{attribute 'GeneratedUsingTerminal: EK1122-0000-0018'}
{attribute addProperty BoxType "EK1122-0000-0018"}
{attribute addProperty Id "Beckhoff_EP5xxxsub_EK1100EK1100_1FC0878B2A_0001_EP5001_0002_0016EP5001_0B28D08722A_0002_EP5101_0002_0016EP5101_87AC78CF32A_0003_EP5101_0002_0017EP5101_87AC78CF32A_0004_EP5101_0002_0018EP5101_87AC78CF32A_0005_EP5101_0002_0019EP5101_87AC78CF32A_0006_EP5101_0011_0016EP5101_7476E94838A_0007_EP5101_0011_0017EP5101_7476E94838A_0008_EP5101_0011_0018EP5101_7476E94838A_0009_EP5101_0011_0019EP5101_7476E94838A_0010_EP5101_1002_0017EP5101_87AC78CF32A_0011_EP5151_0002_0018EP5151_7476E94838A_0012_EP5101_2011_0016EP5101_382A92AF35"}
{attribute addProperty CRC "1751390652"}
{attribute addProperty Size "409"}
TYPE Beckhoff_EP5xxxEK1122_686419BC EXTENDS EK1122_1FC0878B :
STRUCT
	{attribute addProperty Name "Beckhoff_EP5xxxsub_EK1100"}
	{attribute addProperty PreviousPort "Beckhoff EP5xxxEK1122 : D"}
	Beckhoff_EP5xxxsub_EK1100 : EK1100_1FC0878B;
	{attribute addProperty Name "A_0001_EP5001_0002_0016"}
	{attribute addProperty PreviousPort "Beckhoff EP5xxxsub EK1100 : C"}
	A_0001_EP5001_0002_0016 : EP5001_0B28D087;
	{attribute addProperty Name "A_0002_EP5101_0002_0016"}
	{attribute addProperty PreviousPort "A_0001(EP5001-0002-0016) : B"}
	A_0002_EP5101_0002_0016 : EP5101_87AC78CF;
	{attribute addProperty Name "A_0003_EP5101_0002_0017"}
	{attribute addProperty PreviousPort "A_0002(EP5101-0002-0016) : B"}
	A_0003_EP5101_0002_0017 : EP5101_87AC78CF;
	{attribute addProperty Name "A_0004_EP5101_0002_0018"}
	{attribute addProperty PreviousPort "A_0003(EP5101-0002-0017) : B"}
	A_0004_EP5101_0002_0018 : EP5101_87AC78CF;
	{attribute addProperty Name "A_0005_EP5101_0002_0019"}
	{attribute addProperty PreviousPort "A_0004(EP5101-0002-0018) : B"}
	A_0005_EP5101_0002_0019 : EP5101_87AC78CF;
	{attribute addProperty Name "A_0006_EP5101_0011_0016"}
	{attribute addProperty PreviousPort "A_0005(EP5101-0002-0019) : B"}
	A_0006_EP5101_0011_0016 : EP5101_7476E948;
	{attribute addProperty Name "A_0007_EP5101_0011_0017"}
	{attribute addProperty PreviousPort "A_0006(EP5101-0011-0016) : B"}
	A_0007_EP5101_0011_0017 : EP5101_7476E948;
	{attribute addProperty Name "A_0008_EP5101_0011_0018"}
	{attribute addProperty PreviousPort "A_0007(EP5101-0011-0017) : B"}
	A_0008_EP5101_0011_0018 : EP5101_7476E948;
	{attribute addProperty Name "A_0009_EP5101_0011_0019"}
	{attribute addProperty PreviousPort "A_0008(EP5101-0011-0018) : B"}
	A_0009_EP5101_0011_0019 : EP5101_7476E948;
	{attribute addProperty Name "A_0010_EP5101_1002_0017"}
	{attribute addProperty PreviousPort "A_0009(EP5101-0011-0019) : B"}
	A_0010_EP5101_1002_0017 : EP5101_87AC78CF;
	{attribute addProperty Name "A_0011_EP5151_0002_0018"}
	{attribute addProperty PreviousPort "A_0010(EP5101-1002-0017) : B"}
	A_0011_EP5151_0002_0018 : EP5151_7476E948;
	{attribute addProperty Name "A_0012_EP5101_2011_0016"}
	{attribute addProperty PreviousPort "A_0011(EP5151-0002-0018) : B"}
	A_0012_EP5101_2011_0016 : EP5101_382A92AF;
END_STRUCT
END_TYPE

(* stored: Version 1.2.0.0, ProductVersion 3.1.4024.9
   DUT Beckhoff_EP5xxxEK1122_686419BC: Id {6e71dece-0b66-4c86-973a-c23c1cd75295} *)
